FUNCTION_BLOCK read_geophone
VAR_INPUT
	// none
END_VAR
VAR_OUTPUT
	velX : LREAL; // left -> right
	velY : LREAL; // back -> front
	velZ : LREAL; // top -> bottom
END_VAR
VAR
	c1Sample AT %I* : DINT; // channel 1 voltage (mV) -  z axis
	c2Sample AT %I* : DINT; // channel 2 voltage (mV) -  y axis
	c3Sample AT %I* : DINT; // channel 3 voltage (mV) -  x axis
	
	sens : REAL := 78.9; // volts per meter per second
END_VAR

velX := DINT_TO_LREAL(c3Sample) / (sens * 1000);
velY := DINT_TO_LREAL(c2Sample) / (sens * 1000);
velZ := DINT_TO_LREAL(c1Sample) / (sens * 1000);

END_FUNCTION_BLOCK

(* stored: Version 1.1.0.1, ProductVersion 3.1.4024.13
   POU read_geophone: Id {56b7d18b-71f0-4c3f-9840-fefa8f0a6997}, SpecialFunc None *)
